// TIA Portal V19 export
ORGANIZATION_BLOCK "RACK_FLT"   // OB86, STL, RackOrStationFailure
TITLE = "Loss Of Rack Fault"
{ S7_Optimized_Access := 'TRUE' }
   VAR_INPUT
      LADDR : HW_DEVICE;   // Hardware identifier
      Event_Class : Byte;   // Event class
      Fault_ID : Byte;   // Fault identifier
   END_VAR
   VAR_TEMP
      OB86_RACKS_FLTD : Array[0..31] of Bool;
      OB86_DATE_TIME : Date_And_Time;   // Date and time OB86 started
   END_VAR
BEGIN
END_ORGANIZATION_BLOCK
